// Mitsubishi GX Works2 project: 스캔   PLC: Q02/Q02H

PROGRAM MAIN
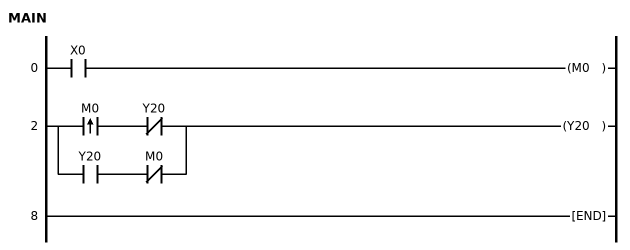
0     LD      X0
      OUT     M0
2     LDP     M0
      ANI     Y20
      LD      Y20
      ANI     M0
      ORB
      OUT     Y20
8     END
END_PROGRAM
